// TIA Portal project "step_motoru_test_modunda_calistirma" (V18)

(* hardware
DEVICE "S7-1200 station_1"  S7-1200 Station
   slot 0: "Rack_0"  S7-1200 Rack  Rack  V1.0
   slot 1: "PLC_1"  CPU 1214C DC/DC/DC  6ES7 214-1AG40-0XB0  V4.6
DEVICE "PC station"  SIMATIC PC station
   slot 0: "PC station"  Rail  SIMATIC PC-Station  V1.0
      slot 125: "Stationmanager"  Station_Manager  V6.0.4
   slot 1: "HMI_RT_1"  WinCC RT Advanced  6AV2 104-0xxxx-xxxx  17.0.0.0
      slot 33792: "Computer interface"  Host interface
*)

// ===== PLC "PLC_1"  CPU 1214C DC/DC/DC =====

VAR_GLOBAL   // PLC tag table "Default tag table"
   "Axis_1_Pulse" AT %Q0.0 : Bool;
   "Axis_1_Direction" AT %Q0.1 : Bool;
   "Axis_1_DriveEnable" AT %Q0.2 : Bool;
   "Axis_1_LowHwLimitSwitch" AT %I0.0 : Bool;
   "Axis_1_HighHwLimitSwitch" AT %I0.1 : Bool;
   "SİSTEM START" AT %I0.2 : Bool;
   "RESET" AT %I0.3 : Bool;
   "BAŞLANGIÇ NOKTASINA HAREKET" AT %I0.4 : Bool;
   "HAREKETİ SONLANDIRIR" AT %I0.5 : Bool;
   "HAREKET BAŞLAT" AT %I0.6 : Bool;
   "HEDEFE GİT" AT %I0.7 : Bool;
   "Tag_1" AT %M0.0 : Bool;
   "YÖN KONTROL" AT %M0.1 : Bool;
   "İLERİ" AT %M0.2 : Bool;
   "GERİ" AT %M0.3 : Bool;
   "FONKSİYON AKTİF" AT %M1.0 : Bool;
   "HIZLANMA SÜRESİ DEĞİŞTİR" AT %M1.1 : Bool;
   "YAVAŞLAMA SÜRESİ DEGİSTİR" AT %M1.2 : Bool;
   "ACİL STOP DEĞİŞTİRME" AT %M1.3 : Bool;
   "SARSINTI YUMUŞATMA DEĞİŞTİRME" AT %M1.4 : Bool;
END_VAR

DATA_BLOCK "STEP KONTROL"   // DB1, Motion_DB
{ S7_Optimized_Access := 'TRUE' }
AUTHOR : SIMATIC
FAMILY : BasicMC
NAME : TO_PTO
VERSION : 2.0
// stored: InstanceOfName TO_Axis_PTO
"TO_Axis_PTO"
BEGIN
   // Axis.PositionLimitsMax_AddressCU = %I0.1
   // Axis.PositionLimitsMin_AddressCU = %I0.0
   // Axis.EnableOutput_AddressCU = %Q0.2
   // Axis.DirectionHwcnAddressCU = %Q0.1
   // Axis.PulseHwcnAddressCU = %Q0.0
   // Pulse.MinDeltaDeltaFrequencyCU = 0.004
   // Pulse.MaxDeltaDeltaFrequencyCU = 1.0E+10
   // Pulse.MinDeltaFrequencyCU = 0.005
   // Pulse.MaxDeltaFrequencyCU = 9.5E+9
   // Pulse.MinFrequencyCU = 1.0
   // Pulse.MaxFrequencyCU = 100000.0
   // Pulse.OutputSourceCU = 16#0000_0000
   // Axis.SelectPTO = 0
END_DATA_BLOCK

ORGANIZATION_BLOCK "Main"   // OB1, LAD, ProgramCycle
TITLE = "Main Program Sweep (Cycle)"
{ S7_Optimized_Access := 'TRUE' }
VERSION : 0.1
// STOPMODE motorun hareketinin ne şekilde sonlanacağını söyler
// 0 ise durma yavaşlayarak gerçekleşir
// 1 ise durma işlemi anında gerçekleşir
// 2 ise durma yavaşlama ile birlikte ayarlanan sarsıntıyı azaltma işelmini de dahil eder
   VAR_INPUT
      Initial_Call : Bool;   // Initial call of this OB
      Remanence : Bool;   // =True, if remanent data are available
   END_VAR
BEGIN

REGION Network 1
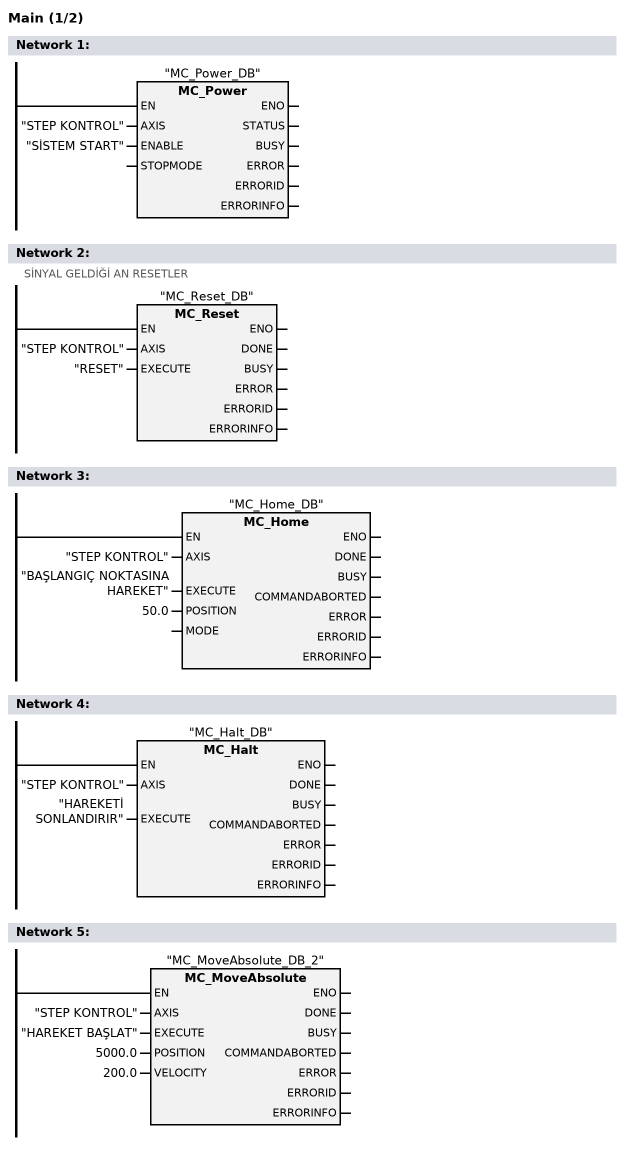
   "MC_Power_DB"(Axis := "STEP KONTROL", Enable := "SİSTEM START");   // MC_Power
END_REGION

REGION Network 2
   // SİNYAL GELDİĞİ AN RESETLER
   "MC_Reset_DB"(Axis := "STEP KONTROL", Execute := "RESET");   // MC_Reset
END_REGION

REGION Network 3
   "MC_Home_DB"(Axis := "STEP KONTROL", Execute := "BAŞLANGIÇ NOKTASINA HAREKET", Position := 50.0);   // MC_Home
END_REGION

REGION Network 4
   "MC_Halt_DB"(Axis := "STEP KONTROL", Execute := "HAREKETİ SONLANDIRIR");   // MC_Halt
END_REGION

REGION Network 5
   "MC_MoveAbsolute_DB_2"(Axis := "STEP KONTROL",   // MC_MoveAbsolute
                          Execute := "HAREKET BAŞLAT",
                          Position := 5000.0,
                          Velocity := 200.0);
END_REGION

REGION Network 6
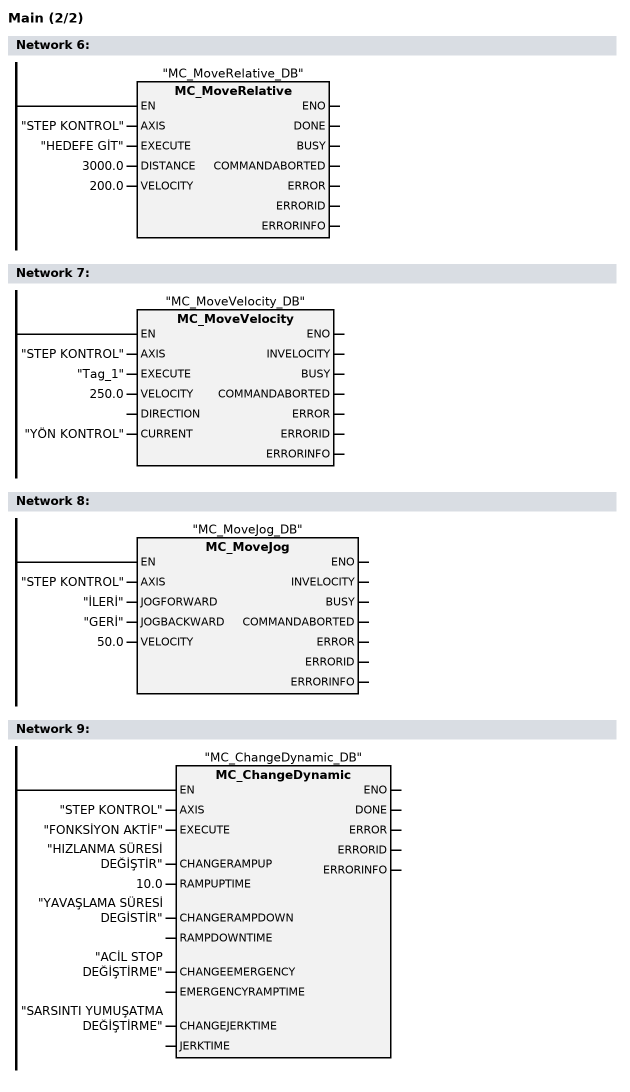
   "MC_MoveRelative_DB"(Axis := "STEP KONTROL", Execute := "HEDEFE GİT", Distance := 3000.0, Velocity := 200.0);   // MC_MoveRelative
END_REGION

REGION Network 7
   "MC_MoveVelocity_DB"(Axis := "STEP KONTROL", Execute := "Tag_1", Velocity := 250.0, Current := "YÖN KONTROL");   // MC_MoveVelocity
END_REGION

REGION Network 8
   "MC_MoveJog_DB"(Axis := "STEP KONTROL", JogForward := "İLERİ", JogBackward := "GERİ", Velocity := 50.0);   // MC_MoveJog
END_REGION

REGION Network 9
   "MC_ChangeDynamic_DB"(Axis := "STEP KONTROL",   // MC_ChangeDynamic
                         Execute := "FONKSİYON AKTİF",
                         ChangeRampUp := "HIZLANMA SÜRESİ DEĞİŞTİR",
                         RampUpTime := 10.0,
                         ChangeRampDown := "YAVAŞLAMA SÜRESİ DEGİSTİR",
                         ChangeEmergency := "ACİL STOP DEĞİŞTİRME",
                         ChangeJerkTime := "SARSINTI YUMUŞATMA DEĞİŞTİRME");
END_REGION
END_ORGANIZATION_BLOCK

(* ===== HMI "HMI_RT_1" =====
system functions are stored by id; their names below are inferred from use
connection "HMI_Connection_1": ETHERNET, S7_1200_OMS

HMI tags "Default tag table"
   "İLERİ" : Bool = PLC İLERİ AT %M0.2, 1 s
   "GERİ" : Bool = PLC GERİ AT %M0.3, 1 s
   "Tag_1" : Bool = PLC Tag_1 AT %M0.0, 1 s

screen "Screen_1" 1024x768
   Button "Button_1" at 55,61 size 96x32; TextOff 'İLERİ'
      on Click: InvertBit("İLERİ")
   Button "Button_2" at 210,61 size 96x32; TextOff 'GERİ'
      on Click: InvertBit("GERİ")
   Button "Button_3" at 58,154 size 96x32; TextOff 'SÜREKLİ'
      on Click: InvertBit("Tag_1")
*)